{attribute addProperty BoxType "EL6690-0001-0000"}
{attribute addProperty Id "StatusAT %I*Status_93A34D63810InputsEMPTY_STRUCTURE000OutputsEMPTY_STRUCTURE000WcStateAT %I*WcState_F855686C1620InfoDataAT %I*InfoData_BC63D37F80100"}
{attribute addProperty CRC "94042852"}
{attribute addProperty SizeInBites "104"}
{attribute addProperty SizeInBytes "13"}
TYPE EL6690_108834A4 :
STRUCT
	{attribute addProperty Name "Status"}
	Status : Status_93A34D63;
	{attribute addProperty Name "Inputs"}
	Inputs : EMPTY_STRUCTURE;
	{attribute addProperty Name "Outputs"}
	Outputs : EMPTY_STRUCTURE;
	{attribute addProperty Name "WcState"}
	WcState : WcState_F855686C;
	{attribute addProperty Name "InfoData"}
	InfoData : InfoData_BC63D37F;
END_STRUCT
END_TYPE

(* stored: Version 1.2.0.0, ProductVersion 3.1.4024.9
   DUT EL6690_108834A4: Id {c52e06cc-dbc6-40af-83cd-3ea79ad8fbdc} *)
